INTERFACE I_CSVEventStorage

METHOD StoreEvent
VAR_INPUT
	stEvent : ST_Event;
END_VAR
END_METHOD

END_INTERFACE

(* stored: Version 1.1.0.1, ProductVersion 3.1.4024.9
   Itf I_CSVEventStorage: Id {1e0e33f4-713c-4e83-82e8-e09af57ab57f}
   Method StoreEvent: Id {94b4fd0d-06ca-4453-a47c-75dcbba0311e} *)
